(* CoDeSys 2.3 export: BUTTONTRIGGEREDSHADER.EXP *)

(* POU Components/Shader/ButtonTriggeredShader, ST *)
FUNCTION_BLOCK ButtonTriggeredShader
VAR_INPUT
	input:BOOL;
END_VAR
VAR_OUTPUT
	closeOut:BOOL;
	openOut:BOOL;
END_VAR
VAR
	Button:Button;
END_VAR
VAR_IN_OUT
	Shader:Shader;
END_VAR
button(input:=input);
shader(switch:= button.fallingEdge);

closeOut:= shader.closing;
openOut:= shader.opening;
END_FUNCTION_BLOCK
